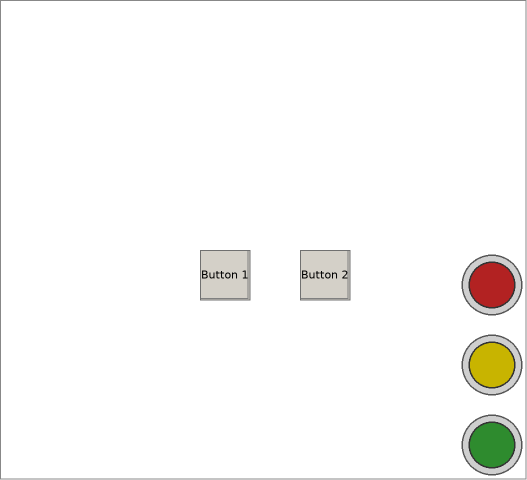
VISUALIZATION Visualization  // 527x480
    Button (200,250 50x50), "Button 1"
        OnMouseClick: toggle MAIN._Button1
    Button (300,250 50x50), "Button 2"
        OnMouseClick: toggle MAIN._Button2
    Lamp1 (457,250 70x70), variable: MAIN._LampR, style: Lamp-Lamp1-Red
    Lamp1 (457,330 70x70), variable: MAIN._LampY, style: Lamp-Lamp1-Yellow
    Lamp1 (457,410 70x70), variable: MAIN._LampG, style: Lamp-Lamp1-Green
END_VISUALIZATION

(* stored: Version 1.1.0.1
   Visu Visualization: Id {e28f008e-7928-4a76-907a-a3c268eb55bb} *)
